Staubli VAL3: onF4Event.pgx

program onF4Event()
  local string l_sMessage
  local bool l_bImport
  local string l_sPath[2]
  local num l_nLocal
  local num l_nKey
  local bool l_bDone
  local num l_nOldValue[4]
  local string l_sButton[2]
  local string l_sItem
begin
  // look if the bButton is enable
  if bButton[3]

    //
  endIf
end
